(* IEC 61131-3 sources: eCockpitGit/test_project/src/%PLC%PLCTest2/%PLOG%Plc Logic/%APP%APP1_Test/%F%NormalFolder/%GVL%GVL_test_1/%PRO%PropAlop_2, 1 file *)

(* ---- %GETSET%Get.st ---- *)
VAR
	temp4:		STRING;
END_VAR

(*%!%__DELIMITER__%!%*)
PropAlop_2		:=		variablssss3;
PropAlop_2		:=		temp4;
